// TIA Portal V16 export
// export: Created 2025-05-24T14:07:57.0082385Z, ExportSetting WithDefaults, DisplayName Totally Integrated Automation Portal, DisplayVersion V16, DisplayName TIA Portal Version Control Interface, DisplayVersion V16, DisplayName TIA Portal Openness, DisplayVersion V16, DisplayName STEP 7 Professional, DisplayVersion V16, DisplayName STEP 7 Safety, DisplayVersion V16, DisplayName WinCC Advanced, DisplayVersion V16
DATA_BLOCK "Ouput_Function_1_Valve1"   // DB19
VERSION : 0.1
// stored: AutoNumber true, InstanceOfName Ouput_Function_1, InstanceOfType FB
"Ouput_Function_1"
   // VAR_INPUT
   //    "Stop Contact" : Bool;
   //    "Manual Command" : Bool;
   //    "Auto Command" : Bool;
   //    "Option Command" : Bool;
   //    "Disable Command" : Bool;
   // END_VAR
   // VAR_OUTPUT
   //    "Ouput Signal" : Bool;
   // END_VAR
BEGIN
END_DATA_BLOCK
